(* PLC project TestBenchEmergency.project, CODESYS CODESYS V3.5 SP19 Patch 1 *)
(* stored: creationDateTime 2026-07-30T21:00:24.172299, modificationDateTime 2026-07-30T21:00:24.172299 *)

(* ═══════════════════════════════════════════════════════════════ ⚙️ ST_EmergencyManagementCmd — Structure de commande interne ─────────────────────────────────────────────────────────────── 📄 Transporte les ordres logiques entre le bloc de décision et le bloc de sortie de la boucle d'urgence. 🏷️ Renommé PowerCutOff_X_Cmd → MaintainA/B_Cmd (polarité maintien : TRUE = voie maintenue saine, FALSE = coupure demandée — la règle C1 interdit un nom portant « coupure » quand le sens est « maintien »). ═══════════════════════════════════════════════════════════════ 📄 Docs : DOC/AF_Partie-01_Analyse_Fonctionnelle_v2.0.md DOC/AF_Partie-01_Analyse_Fonctionnelle_v2.0.md *)
TYPE ST_EmergencyManagementCmd : STRUCT
  MaintainA_Cmd : BOOL;  (* Ordre maintien canal A (TRUE = voie maintenue, FALSE = coupure demandée) *)
  MaintainB_Cmd : BOOL;  (* Ordre maintien canal B (TRUE = voie maintenue, FALSE = coupure demandée) *)
  ArmPulse_Cmd : BOOL;  (* Ordre impulsion de réarmement (TRUE = bobine réarmement activée) *)
END_STRUCT;
END_TYPE

(* ═══════════════════════════════════════════════════════════════ 🚦 ST_State_Emergency — État public de la chaîne d'arrêt d'urgence ─────────────────────────────────────────────────────────────── 📄 Produit par FB_Safety_EmergencyManagement (sortie State). Consommé par PRG_09_Supervision → GVL_IHM.Modes.State pour IHM, et par GVL_Troubleshooting pour diagnostic. 🎯 Champs lecture seule — aucun lecteur n'est autorisé à l'écrire. ═══════════════════════════════════════════════════════════════ 📄 Docs : DOC/AF_Partie-01_Analyse_Fonctionnelle_v2.0.md DOC/AF_Partie-01_Analyse_Fonctionnelle_v2.0.md §8.2 *)
TYPE ST_State_Emergency : STRUCT
  ChainOk : BOOL;  (* 🔗 Boucle AU fermée (EmergencyChainClosed_DI = TRUE) *)
  ContactorOk : BOOL;  (* 🔌 Contacteur puissance confirmé engagé (PowerContactorEngaged_DI = TRUE) *)
  Step : INT;  (* 🔢 Étape séquence armement : 0=IDLE, 1=TestA, 2=RestoreA, 3=TestB, 4=RestoreB, 5=Pulse, 6=Confirm *)
  Armable : BOOL;  (* 🟢 Réarmement possible maintenant : chain OK, step=0, pas de lockout, pas de redondance échouée, pas de contacteur déjà engagé *)
  ArmingBusy : BOOL;  (* ⏳ Séquence armement OU lockout en cours (nouvelle demande ignorée) *)
END_STRUCT;
END_TYPE

(* ═══════════════════════════════════════════════════════════════ 🛡️ ST_Diag_Emergency — Diagnostic et erreurs de la chaîne AU ─────────────────────────────────────────────────────────────── 📄 Produit par FB_Safety_EmergencyManagement (sortie Diag). Consommé par PRG_09_Supervision et GVL_Troubleshooting. 🎯 Champs lecture seule — producteur unique = FB composite. ═══════════════════════════════════════════════════════════════ 📄 Docs : DOC/AF_Partie-01_Analyse_Fonctionnelle_v2.0.md DOC/AF_Partie-01_Analyse_Fonctionnelle_v2.0.md §8.2 *)
TYPE ST_Diag_Emergency : STRUCT
  Error : BOOL;  (* 🔴 Synthèse : (ErrorId <> 0) *)
  ErrorId : WORD;  (* ❌ bit0 = RedundancyTestFailed (auto-test A/B), bit1 = EmergencyArmingFailed (timeout confirm contacteur) *)
  RedundancyTestFailed : BOOL;  (* 🔴 Canal A ou B resté collé/shunté détecté à l'auto-test — Reset requis (cause disparue) *)
  ArmFailed : BOOL;  (* 🔴 Impulsion envoyée mais contacteur puissance non confirmé sous 2 s — Reset + contacteur engagé requis *)
  LockoutActive : BOOL;  (* ⏳ Verrouillage temporel de 5 s entre tentatives de réarmement échouées *)
END_STRUCT;
END_TYPE

{attribute 'qualified_only'}
VAR_GLOBAL RETAIN  (* GVL_PERSISTENT_AU - ═══════════════════════════════════════════════════════════════ 💾 GVL_PERSISTENT_AU — Variables persistantes chaîne AU ─────────────────────────────────────────────────────────────── 📄 Rôle : Regroupe les réglages persistants RETAIN propres au domaine Arrêt d'Urgence (FB_Safety_EmergencyManagement). 🎯 Objectif : dissocier les réglages AU des autres domaines (treuils, benne, cycle, etc.) pour les bundles de test. 🔒 RETAIN : survit aux arrêts/redémarrages PLC. ═══════════════════════════════════════════════════════════════ 📄 Docs : DOC/AF_Partie-01_Analyse_Fonctionnelle_v2.0.md DOC/AF_Partie-01_Analyse_Fonctionnelle_v2.0.md *)
  TonTestDuration : TIME := TIME#200ms;  (* ⏱️ Temporisations de la séquence de réarmement (AF §3.5) Les valeurs ci-dessous sont les défauts de la spec. Ne pas modifier sans comprendre la séquence complète (auto-test A/B). Test/Restore A ou B *)
  TonArmingPulseDuration : TIME := TIME#1s0ms;  (* Impulsion de réarmement *)
  TonArmingConfirmTimeout : TIME := TIME#2s0ms;  (* Timeout confirmation contacteur *)
  TonArmingLockout : TIME := TIME#5s0ms;  (* Verrouillage anti-réessai *)
  CfgEmergencyChainNormallyClosed : BOOL := TRUE;  (* 🛡️ Configuration chaîne AU TRUE = boucle AU fermée = sain *)
  CfgContactorNormallyOpen : BOOL := TRUE;  (* TRUE = contacteur engagé = sain *)
END_VAR

{attribute 'qualified_only'}
VAR_GLOBAL  (* GVL_Simulation_AU - ═══════════════════════════════════════════════════════════════ 🧪 GVL_Simulation_AU — Simulation hardware pour test chaîne AU ─────────────────────────────────────────────────────────────── 📄 Remplace les signaux physiques réels (DI/Q) pour le test en isolation de FB_Safety_EmergencyManagement. 🎯 Pattern identique à GVL_Simulation (projet réel) : domaine SimMachineActive = simulation AU. Polarité : TRUE = simulé, FALSE = réel. ═══════════════════════════════════════════════════════════════ 📄 Docs : DOC/AF_Partie-01_Analyse_Fonctionnelle_v2.0.md DOC/AF_Partie-13_Fonction_Simulation_v2.0.md *)
  SimulationModeActive : BOOL := TRUE;  (* 🔑 Bit maître — rien n'est simulé si FALSE *)
  SimChainClosed : BOOL := TRUE;  (* 🛡️ Simulation du matériel AU Simule EmergencyChainClosed_DI fermée *)
  SimContactorEngaged : BOOL := FALSE;  (* Simule retour contacteur puissance *)
  SimPowerCutOffReq : BOOL := FALSE;  (* ⚡ Simulation coupure métier (remplace OR des 3 safety domaines) TRUE = une safety demande la coupure *)
END_VAR

{attribute 'qualified_only'}
VAR_GLOBAL  (* GVL_IHM_AU - ═══════════════════════════════════════════════════════════════ 🖥️ GVL_IHM_AU — Structure IHM pour test chaîne AU ─────────────────────────────────────────────────────────────── 📄 Réplique les champs de ST_ModesCmd/ST_ModesState nécessaires au pilotage de FB_Safety_EmergencyManagement, sans les dépendances aux autres domaines (treuils, translation...). 🎯 Pattern identique à GVL_IHM.Modes.Cmd (projet réel). ═══════════════════════════════════════════════════════════════ 📄 Docs : DOC/AF_Partie-01_Analyse_Fonctionnelle_v2.0.md DOC/AF_Partie-07_Interface_IHM_v2.0.md *)
  BtnEmergencyArming : BOOL;  (* 🎮 Commandes IHM (miroir de ST_ModesCmd) Front demande réarmement contacteur *)
  BtnEmergencyCutOff : BOOL;  (* Niveau coupure IHM maintenue *)
  BtnFaultReset : BOOL;  (* Front acquittement défauts *)
END_VAR

(* ═══════════════════════════════════════════════════════════════ 🛡️ FB_Safety_EmergencyManagement — Bloc Safety Composite (Parent) ─────────────────────────────────────────────────────────────── 📄 Rôle : Bloc de sécurité principal de la boucle d'arrêt d'urgence. 🧩 Encapsule la Logique (FB_Safety_EmergencyManagementLogic) et le Pilote Physique (FB_Safety_EmergencyManagementOutput) par composition. 📤 Produit les bus publics ST_State_Emergency et ST_Diag_Emergency en sortie, consommés par Supervision et Troubleshooting. 🏷️ Renommé PowerCutOff_A/B_RQ → MaintainA/B_RQ (polarité maintien), EmergencyArming_RQ → ArmPulse_RQ (cohérence nommage). ═══════════════════════════════════════════════════════════════ 📄 Docs : DOC/AF_Partie-01_Analyse_Fonctionnelle_v2.0.md DOC/AF_Partie-01_Analyse_Fonctionnelle_v2.0.md DOC/AF_Partie-03_Contrats_Composants_v2.0.md *)
FUNCTION_BLOCK FB_Safety_EmergencyManagement
  VAR_INPUT
    Enable : BOOL;  (* Active la surveillance *)
    Reset : BOOL;  (* Front acquittement défauts *)
    ArmRequest : BOOL;  (* Demande de réarmement (BtnEmergencyArming) *)
    EmergencyChainClosed : BOOL;  (* Retour physique boucle d'urgence amont contacteur *)
    PowerContactorEngaged : BOOL;  (* Confirmation contacteur de puissance principal *)
    PowerCutOffRequest : BOOL;  (* Requête de coupure logique issue des métiers *)
    BtnEmergencyCutOff : BOOL;  (* Commande d'ouverture d'urgence depuis l'IHM *)
  END_VAR
  VAR_OUTPUT
    Ready : BOOL;
    Busy : BOOL;
    Done : BOOL;
    Error : BOOL;
    ErrorId : WORD;  (* bit0: RedundancyTestFailed, bit1: EmergencyArmingFailed, bit3: StartupFail *)
    MaintainA_RQ : BOOL;  (* ⚡ Sorties physiques — renommées (polarité maintien explicite) Sortie de pilotage canal A (TRUE = voie maintenue, FALSE = coupure) *)
    MaintainB_RQ : BOOL;  (* Sortie de pilotage canal B (TRUE = voie maintenue, FALSE = coupure) *)
    ArmPulse_RQ : BOOL;  (* Impulsion réarmement physique (1s) *)
    State : ST_State_Emergency;  (* 🚦 Bus d'état public (AF §8.2) ChainOk, ContactorOk, Step, Armable, ArmingBusy *)
    Diag : ST_Diag_Emergency;  (* Error, ErrorId, Redundancy, ArmFailed, Lockout *)
    ArmingSeqStep : INT;  (* 🩺 Diagnostics scalaires (rétrocompatibilité PRG_10/GVL_Global) *)
    RedundancyTestFailed : BOOL;
    EmergencyArmingFailed : BOOL;
    EmergencyArmingLockoutActive : BOOL;
  END_VAR
  VAR
    Logic : FB_Safety_EmergencyManagementLogic;  (* 🧱 Composition interne des sous-blocs *)
    Output : FB_Safety_EmergencyManagementOutput;
  END_VAR

            

// === IMPLEMENTATION ===

// 🛑 1. Appels des instances internes
Logic(
    Enable := Enable,
    Reset := Reset,
    ArmRequest := ArmRequest,
    EmergencyChainClosed := EmergencyChainClosed,
    PowerContactorEngaged := PowerContactorEngaged,
    PowerCutOffRequest := PowerCutOffRequest,
    BtnEmergencyCutOff := BtnEmergencyCutOff
);

Output(
    Enable := Enable,
    Cmd := Logic.Cmd,
    ChainOk := EmergencyChainClosed,
    ContactorOk := PowerContactorEngaged,
    ArmingStep := Logic.ArmingSeqStep,
    Armable := Logic.Armable,
    ArmingBusy := Logic.ArmingBusy,
    Error := Logic.Error,
    ErrorId := Logic.ErrorId,
    RedundancyTestFailed := Logic.RedundancyTestFailed,
    ArmFailed := Logic.EmergencyArmingFailed,
    LockoutActive := Logic.EmergencyArmingLockoutActive
);

// 📤 2. Propagation des signaux vers les sorties du bloc parent
Ready := Enable AND NOT Logic.StartupFail;
Busy  := (Logic.ArmingSeqStep <> 0) OR Logic.EmergencyArmingLockoutActive;
Done  := PowerContactorEngaged;
Error := Logic.Error;
ErrorId := Logic.ErrorId;

// ⚡ Sorties physiques
MaintainA_RQ   := Output.MaintainA_RQ;
MaintainB_RQ   := Output.MaintainB_RQ;
ArmPulse_RQ    := Output.ArmPulse_RQ;

// 🚦 Bus publics
State := Output.State;
Diag  := Output.Diag;

// 🩺 Diagnostics scalaires (rétrocompatibilité)
ArmingSeqStep                := Logic.ArmingSeqStep;
RedundancyTestFailed         := Logic.RedundancyTestFailed;
EmergencyArmingFailed        := Logic.EmergencyArmingFailed;
EmergencyArmingLockoutActive := Logic.EmergencyArmingLockoutActive;

          
END_FUNCTION_BLOCK

(* ═══════════════════════════════════════════════════════════════ 🛡️ FB_Safety_EmergencyManagementLogic — Décision & Séquencement ─────────────────────────────────────────────────────────────── 📄 Rôle : Gère la machine d'état d'auto-test et de réarmement de la boucle d'arrêt d'urgence. Produit les consignes logiques et les bus d'état/diagnostic. 🏷️ Renommé PowerCutOff_X_Cmd → MaintainA/B_Cmd (polarité maintien). Ajout autotest démarrage (§5.4 AF01) + bus State/Diag. ═══════════════════════════════════════════════════════════════ 📄 Docs : DOC/AF_Partie-01_Analyse_Fonctionnelle_v2.0.md DOC/AF_Partie-01_Analyse_Fonctionnelle_v2.0.md DOC/AF_Partie-03_Contrats_Composants_v2.0.md *)
FUNCTION_BLOCK FB_Safety_EmergencyManagementLogic
  VAR_INPUT
    Enable : BOOL;  (* Active la surveillance *)
    Reset : BOOL;  (* Front acquittement défauts *)
    ArmRequest : BOOL;  (* Demande de réarmement (BtnEmergencyArming) *)
    EmergencyChainClosed : BOOL;  (* Retour physique boucle d'urgence amont contacteur *)
    PowerContactorEngaged : BOOL;  (* Confirmation contacteur de puissance principal *)
    PowerCutOffRequest : BOOL;  (* Requête de coupure logique issue des métiers *)
    BtnEmergencyCutOff : BOOL;  (* Commande d'ouverture d'urgence depuis l'IHM *)
  END_VAR
  VAR_OUTPUT
    Error : BOOL;
    ErrorId : WORD;  (* bit0: RedundancyTestFailed, bit1: EmergencyArmingFailed *)
    Cmd : ST_EmergencyManagementCmd;  (* Structure de commande logique produite *)
    ArmingSeqStep : INT;  (* Étape de diagnostic : 0=IDLE, 1=TestA, 2=RestoreA, 3=TestB, 4=RestoreB, 5=Pulse, 6=Confirm *)
    RedundancyTestFailed : BOOL;  (* Canal A ou B resté collé/shunté détecté à l'auto-test *)
    EmergencyArmingFailed : BOOL;  (* Contacteur de puissance n'a pas confirmé l'armement *)
    EmergencyArmingLockoutActive : BOOL;  (* Verrouillage temporel de 5s entre les essais *)
    Armable : BOOL;  (* 🆕 Bus State/Diag internes — repris par le composite pour les DUT publics 🟢 Réarmement possible maintenant *)
    ArmingBusy : BOOL;  (* ⏳ Séquence ou lockout en cours *)
    StartupFail : BOOL;  (* 🔴 Autotest démarche échoué *)
  END_VAR
  VAR
    ResetEdge : R_TRIG;
    ArmReqEdge : R_TRIG;
    EnableRising : R_TRIG;
    ForceTestA : BOOL;
    ForceTestB : BOOL;
    TonTestA : TON;
    TonRestoreA : TON;
    TonTestB : TON;
    TonRestoreB : TON;
    TonArmingPulse : TON;
    TonArmingConfirm : TON;
    TonArmingLockout : TON;
    StartupCheckDone : BOOL;  (* 🆕 Autotest démarrage TRUE = autotest passé, attente réarmement *)
    StartupCheckOK : BOOL;  (* Résultat autotest (latche le temps du front) *)
  END_VAR

            

// === IMPLEMENTATION ===

// 🔄 Fronts
EnableRising(CLK := Enable);
ResetEdge(CLK := Reset);
ArmReqEdge(CLK := ArmRequest);

// 🛑 1. GATE — neutralisation si désactivé
IF NOT Enable THEN
    Error := FALSE;
    ErrorId := 16#0000;
    Cmd.MaintainA_Cmd := FALSE;
    Cmd.MaintainB_Cmd := FALSE;
    Cmd.ArmPulse_Cmd := FALSE;
    ArmingSeqStep := 0;
    RedundancyTestFailed := FALSE;
    EmergencyArmingFailed := FALSE;
    EmergencyArmingLockoutActive := FALSE;
    ForceTestA := FALSE;
    ForceTestB := FALSE;
    Armable := FALSE;
    ArmingBusy := FALSE;
    StartupFail := FALSE;
    StartupCheckDone := FALSE;
    StartupCheckOK := FALSE;
    TonTestA(IN := FALSE);
    TonRestoreA(IN := FALSE);
    TonTestB(IN := FALSE);
    TonRestoreB(IN := FALSE);
    TonArmingPulse(IN := FALSE);
    TonArmingConfirm(IN := FALSE);
    TonArmingLockout(IN := FALSE);
    RETURN;
END_IF;

// 🏁 2. AUTOTEST DÉMARRAGE (§5.4 AF01)
// Vérifications synchrones 1 cycle au premier passage Enable=TRUE
IF EnableRising.Q THEN
    StartupCheckDone := FALSE;
END_IF;

IF NOT StartupCheckDone THEN
    // Exécute les 4 contrôles en 1 cycle
    StartupCheckOK := EmergencyChainClosed          // 1. Boucle AU fermée
                      AND NOT PowerContactorEngaged // 2. Contacteur au repos
                      AND (ArmingSeqStep = 0);      // 4. Pas de séquence résiduelle
    // Le maintien A/B est vérifié via l'absence de RedundancyTestFailed
    // (si un canal est ouvert au démarrage, RedundancyTestFailed sera levé
    //  à la première tentative de réarmement — pas bloquant au boot)
    StartupCheckDone := TRUE;
    StartupFail := NOT StartupCheckOK;
    // Si échec : on reste en attente, ErrorId est positionné
    IF NOT StartupCheckOK THEN
        ErrorId := 16#0008; // bit3 = startup autotest fail
        Error := TRUE;
    END_IF;
    RETURN; // 1 cycle pour laisser le temps aux entrées de se stabiliser
ELSE
    StartupFail := FALSE;
END_IF;

// 🔍 3. ACQUITTEMENT DES DÉFAUTS
IF ResetEdge.Q THEN
    RedundancyTestFailed := FALSE;
    StartupFail := FALSE;
    IF PowerContactorEngaged THEN
        EmergencyArmingFailed := FALSE;
    END_IF;
    // Reset efface aussi bit3 d'ErrorId
    ErrorId := ErrorId AND 16#FFF7;
END_IF;

// 🚦 4. DÉCLENCHEMENT DE LA SÉQUENCE DE SÉCURITÉ
IF ArmReqEdge.Q AND (ArmingSeqStep = 0) AND EmergencyChainClosed 
   AND NOT EmergencyArmingLockoutActive 
   AND NOT PowerContactorEngaged THEN
    ArmingSeqStep := 1;
END_IF;

// ⏱️ Étape 1 : Coupe canal A seul, vérifie que la boucle tombe
TonTestA(IN := (ArmingSeqStep = 1), PT := T#200ms);
IF ArmingSeqStep = 1 THEN
    ForceTestA := TRUE;
    IF TonTestA.Q THEN
        ForceTestA := FALSE;
        IF EmergencyChainClosed THEN
            RedundancyTestFailed := TRUE;
            ArmingSeqStep := 0;
        ELSE
            ArmingSeqStep := 2;
        END_IF;
    END_IF;
ELSE
    ForceTestA := FALSE;
END_IF;

// ⏱️ Étape 2 : Restaure A, attend le retour sain de la boucle amont
TonRestoreA(IN := (ArmingSeqStep = 2), PT := T#200ms);
IF (ArmingSeqStep = 2) AND TonRestoreA.Q THEN
    IF EmergencyChainClosed THEN
        ArmingSeqStep := 3;
    ELSE
        ArmingSeqStep := 0;
    END_IF;
END_IF;

// ⏱️ Étape 3 : Coupe canal B seul, vérifie que la boucle tombe
TonTestB(IN := (ArmingSeqStep = 3), PT := T#200ms);
IF ArmingSeqStep = 3 THEN
    ForceTestB := TRUE;
    IF TonTestB.Q THEN
        ForceTestB := FALSE;
        IF EmergencyChainClosed THEN
            RedundancyTestFailed := TRUE;
            ArmingSeqStep := 0;
        ELSE
            ArmingSeqStep := 4;
        END_IF;
    END_IF;
ELSE
    ForceTestB := FALSE;
END_IF;

// ⏱️ Étape 4 : Restaure B, attend le retour sain de la boucle amont
TonRestoreB(IN := (ArmingSeqStep = 4), PT := T#200ms);
IF (ArmingSeqStep = 4) AND TonRestoreB.Q THEN
    IF EmergencyChainClosed THEN
        ArmingSeqStep := 5;
    ELSE
        ArmingSeqStep := 0;
    END_IF;
END_IF;

// ⏱️ Étape 5 : Les 2 canaux validés -> impulsion réarmement physique (1s)
TonArmingPulse(IN := (ArmingSeqStep = 5), PT := T#1s);
Cmd.ArmPulse_Cmd := (ArmingSeqStep = 5);
IF (ArmingSeqStep = 5) AND TonArmingPulse.Q THEN
    ArmingSeqStep := 6;
END_IF;

// ⏱️ Étape 6 : Attente confirmation contacteur principal (2s max)
TonArmingConfirm(IN := (ArmingSeqStep = 6), PT := T#2s);
IF ArmingSeqStep = 6 THEN
    IF PowerContactorEngaged THEN
        ArmingSeqStep := 0;
        EmergencyArmingLockoutActive := FALSE;
    ELSIF TonArmingConfirm.Q THEN
        EmergencyArmingFailed := TRUE;
        ArmingSeqStep := 0;
        EmergencyArmingLockoutActive := TRUE;
    END_IF;
END_IF;

// ⏱️ Séquence de verrouillage temporel (5s)
TonArmingLockout(IN := EmergencyArmingLockoutActive, PT := T#5s);
IF TonArmingLockout.Q THEN
    EmergencyArmingLockoutActive := FALSE;
END_IF;

// 📤 5. GÉNÉRATION DES CONSIGNES LOGIQUES
Cmd.MaintainA_Cmd := NOT PowerCutOffRequest AND NOT ForceTestA AND NOT BtnEmergencyCutOff AND NOT RedundancyTestFailed;
Cmd.MaintainB_Cmd := NOT PowerCutOffRequest AND NOT ForceTestB AND NOT BtnEmergencyCutOff AND NOT RedundancyTestFailed;
// ArmPulse_Cmd déjà positionné à l'étape 5 ci-dessus (garder FALSE hors étape 5)
IF ArmingSeqStep <> 5 THEN
    Cmd.ArmPulse_Cmd := FALSE;
END_IF;

// 🚦 6. ÉTATS PUBLICS (repris par le composite dans State/Diag)
Armable := EmergencyChainClosed
           AND (ArmingSeqStep = 0)
           AND NOT EmergencyArmingLockoutActive
           AND NOT RedundancyTestFailed
           AND NOT PowerContactorEngaged;

ArmingBusy := (ArmingSeqStep <> 0) OR EmergencyArmingLockoutActive;

// 📤 7. SYNTHÈSE DES ERREURS
ErrorId := 16#0000;
IF RedundancyTestFailed THEN
    ErrorId := ErrorId OR 16#0001;
END_IF;
IF EmergencyArmingFailed THEN
    ErrorId := ErrorId OR 16#0002;
END_IF;
// bit3 (16#0008) = StartupFail, positionné au §2 si autotest échoué
// — ne pas l'effacer ici (reset explicite requis)

Error := (ErrorId <> 16#0000);

          
END_FUNCTION_BLOCK

(* ═══════════════════════════════════════════════════════════════ 📤 FB_Safety_EmergencyManagementOutput — Pilote physique + bus état/diag ─────────────────────────────────────────────────────────────── 📄 Rôle : Transmet les ordres de sécurité logiques vers les sorties physiques ET produit les bus d'état et diagnostic publics (ST_State_Emergency / ST_Diag_Emergency). 🧩 Instance privée du composite FB_Safety_EmergencyManagement — jamais appelée hors du composite. ═══════════════════════════════════════════════════════════════ 📄 Docs : DOC/AF_Partie-01_Analyse_Fonctionnelle_v2.0.md DOC/AF_Partie-01_Analyse_Fonctionnelle_v2.0.md *)
FUNCTION_BLOCK FB_Safety_EmergencyManagementOutput
  VAR_INPUT
    Enable : BOOL;  (* Active le pilote (FALSE = toutes sorties à FALSE) *)
    Cmd : ST_EmergencyManagementCmd;  (* Ordres logiques reçus du bloc logique *)
    ChainOk : BOOL;  (* Miroir EmergencyChainClosed (pour bus State) *)
    ContactorOk : BOOL;  (* Miroir PowerContactorEngaged (pour bus State) *)
    ArmingStep : INT;  (* Miroir ArmingSeqStep (pour bus State) *)
    Armable : BOOL;  (* Calculé par Logic (pour bus State) *)
    ArmingBusy : BOOL;  (* Calculé par Logic (pour bus State) *)
    Error : BOOL;  (* Miroir Error (pour bus Diag) *)
    ErrorId : WORD;  (* Miroir ErrorId (pour bus Diag) *)
    RedundancyTestFailed : BOOL;  (* Miroir (pour bus Diag) *)
    ArmFailed : BOOL;  (* Miroir (pour bus Diag) *)
    LockoutActive : BOOL;  (* Miroir (pour bus Diag) *)
  END_VAR
  VAR_OUTPUT
    MaintainA_RQ : BOOL;  (* ⚡ Sorties physiques terminales Vers relais maintien canal A — TRUE = voie maintenue, FALSE = coupure *)
    MaintainB_RQ : BOOL;  (* Vers relais maintien canal B — TRUE = voie maintenue, FALSE = coupure *)
    ArmPulse_RQ : BOOL;  (* Vers contacteur impulsion réarmement — TRUE = pulse actif *)
    State : ST_State_Emergency;  (* 🚦 Bus d'état public *)
    Diag : ST_Diag_Emergency;
  END_VAR

            

// === IMPLEMENTATION ===

IF NOT Enable THEN
    MaintainA_RQ   := FALSE;
    MaintainB_RQ   := FALSE;
    ArmPulse_RQ    := FALSE;

    State.ChainOk        := FALSE;
    State.ContactorOk    := FALSE;
    State.Step           := 0;
    State.Armable        := FALSE;
    State.ArmingBusy     := FALSE;

    Diag.Error                := FALSE;
    Diag.ErrorId              := 16#0000;
    Diag.RedundancyTestFailed := FALSE;
    Diag.ArmFailed            := FALSE;
    Diag.LockoutActive        := FALSE;
    RETURN;
END_IF;

// ⚡ Sorties physiques — écriture directe des ordres logiques
MaintainA_RQ := Cmd.MaintainA_Cmd;
MaintainB_RQ := Cmd.MaintainB_Cmd;
ArmPulse_RQ  := Cmd.ArmPulse_Cmd;

// 🚦 Bus d'état public
State.ChainOk        := ChainOk;
State.ContactorOk    := ContactorOk;
State.Step           := ArmingStep;
State.Armable        := Armable;
State.ArmingBusy     := ArmingBusy;

// 🛡️ Bus diagnostic public
Diag.Error                := Error;
Diag.ErrorId              := ErrorId;
Diag.RedundancyTestFailed := RedundancyTestFailed;
Diag.ArmFailed            := ArmFailed;
Diag.LockoutActive        := LockoutActive;

          
END_FUNCTION_BLOCK

(* ═══════════════════════════════════════════════════════════════ 📥 PRG_AU_Acquisition — Acquisition et qualification des entrées AU ─────────────────────────────────────────────────────────────── 📄 Lit les signaux simulés (GVL_Simulation_AU) ou réels (à connecter sur site) et les qualifie avant de les transmettre au composite. 🧩 Remplit le rôle de PRG_00_Inputs pour le domaine AU uniquement, avec les mêmes structures ST_HwMachine (partielle). 🎯 Pattern : frontière unique HwIn (lot L5 du projet réel). ═══════════════════════════════════════════════════════════════ 📄 Docs : DOC/AF_Partie-01_Analyse_Fonctionnelle_v2.0.md DOC/AF_Partie-06_Acquisition_Qualification_IO_v2.0.md *)
PROGRAM PRG_AU_Acquisition
  VAR_OUTPUT
    EmergencyChainClosed : BOOL;  (* 🔌 Signaux qualifiés vers le reste du programme Boucle AU fermée (qualifié) *)
    PowerContactorEngaged : BOOL;  (* Contacteur puissance engagé (qualifié) *)
    PowerCutOffRequest : BOOL;  (* Demande coupure safety métier (agrégé) *)
    SimActive : BOOL;  (* 🚦 État simulation (pour diagnostic) *)
  END_VAR
  VAR
    TonChainFilter : TON;  (* Anti-rebond logiciel (20 ms, comme PRG_00_Inputs) *)
    TonContactorFilter : TON;
  END_VAR

            

// === IMPLEMENTATION ===

// 🔬 Source : simulé ou réel ?
// En test, on lit depuis GVL_Simulation_AU (SimulationModeActive = TRUE par défaut)
SimActive := GVL_Simulation_AU.SimulationModeActive;

// 🎯 Qualification de la boucle AU (anti-rebond 20 ms)
TonChainFilter(IN := GVL_Simulation_AU.SimChainClosed, PT := T#20ms);
EmergencyChainClosed := TonChainFilter.Q;

// 🎯 Qualification retour contacteur (anti-rebond 20 ms)
TonContactorFilter(IN := GVL_Simulation_AU.SimContactorEngaged, PT := T#20ms);
PowerContactorEngaged := TonContactorFilter.Q;

// 🎯 Agrégation coupure métier (simulée ici, proviendrait de PRG_03_Safety en réel)
PowerCutOffRequest := GVL_Simulation_AU.SimPowerCutOffReq;

          
END_PROGRAM

(* ═══════════════════════════════════════════════════════════════ 📤 PRG_AU_Outputs — Écriture des sorties AU (dernière couche) ─────────────────────────────────────────────────────────────── 📄 Appelle FB_Safety_EmergencyManagement et écrit les variables Q physiques (PowerKeepAlive_A/B_RQ, EmergencyArming_RQ). 🧩 Remplit le rôle de PRG_10_Outputs_LD pour le domaine AU. 🎯 Ordre d'appel obligatoire : PRG_AU_Acquisition → PRG_AU_Outputs (même cycle, même tâche). 🚦 Produit les bus ST_State_Emergency et ST_Diag_Emergency observables en Watch pour vérification de la séquence. ═══════════════════════════════════════════════════════════════ 📄 Docs : DOC/AF_Partie-01_Analyse_Fonctionnelle_v2.0.md DOC/AF_Partie-01_FB_Safety_EmergencyManagement_v1.0.md *)
PROGRAM PRG_AU_Outputs
  VAR_OUTPUT
    PowerKeepAlive_A_RQ : BOOL;  (* ⚡ Sorties physiques terminales (mêmes noms que le projet réel) Relais maintien canal A (TRUE = voie maintenue) *)
    PowerKeepAlive_B_RQ : BOOL;  (* Relais maintien canal B (TRUE = voie maintenue) *)
    EmergencyArming_RQ : BOOL;  (* Impulsion réarmement contacteur (1s) *)
    State : ST_State_Emergency;  (* 🚦 Bus d'état et diagnostic pour observation Watch *)
    Diag : ST_Diag_Emergency;
  END_VAR
  VAR
    instEmergencyManagement : FB_Safety_EmergencyManagement;  (* Instance unique du composite AU *)
  END_VAR

            

// === IMPLEMENTATION ===

// 🛡️ Appel du composite — entrées depuis Acquisition + IHM
instEmergencyManagement(
    Enable := TRUE,
    Reset := GVL_IHM_AU.BtnFaultReset,
    ArmRequest := GVL_IHM_AU.BtnEmergencyArming,
    EmergencyChainClosed := PRG_AU_Acquisition.EmergencyChainClosed,
    PowerContactorEngaged := PRG_AU_Acquisition.PowerContactorEngaged,
    PowerCutOffRequest := PRG_AU_Acquisition.PowerCutOffRequest,
    BtnEmergencyCutOff := GVL_IHM_AU.BtnEmergencyCutOff
);

// ⚡ Sorties physiques
PowerKeepAlive_A_RQ := instEmergencyManagement.MaintainA_RQ;
PowerKeepAlive_B_RQ := instEmergencyManagement.MaintainB_RQ;
EmergencyArming_RQ  := instEmergencyManagement.ArmPulse_RQ;

// 🚦 Observation structurée
State := instEmergencyManagement.State;
Diag  := instEmergencyManagement.Diag;

          
END_PROGRAM

(* ═══════════════════════════════════════════════════════════════ 🧪 PRG_AU_TestBench — Programme principal de test chaîne AU ─────────────────────────────────────────────────────────────── 📄 Ordonnance les étages Acquisition → Outputs dans l'ordre correct (même flux que MainTask réelle). 🎮 Pilotage via Watch CODESYS : GVL_IHM_AU.BtnEmergencyArming = TRUE → lance réarmement GVL_IHM_AU.BtnFaultReset = TRUE → acquitte défauts GVL_IHM_AU.BtnEmergencyCutOff = TRUE → coupure IHM GVL_Simulation_AU.SimContactorEngaged = TRUE → simule retour contacteur GVL_Simulation_AU.SimPowerCutOffReq = TRUE → simule coupure métier 👁️ Observation : PRG_AU_Outputs.State.Step → étape séquence (0..6) PRG_AU_Outputs.PowerKeepAlive_A_RQ → état maintien A PRG_AU_Outputs.EmergencyArming_RQ → pulse réarmement PRG_AU_Outputs.Diag → erreurs/locks ═══════════════════════════════════════════════════════════════ 📄 Docs : DOC/AF_Partie-01_Analyse_Fonctionnelle_v2.0.md DOC/AF_Partie-01_FB_Safety_EmergencyManagement_v1.0.md *)
PROGRAM PRG_AU_TestBench
  VAR_OUTPUT
    StepLabel : STRING;  (* 🩺 Synthèse lisible pour Watch *)
    MaintainA : BOOL;
    MaintainB : BOOL;
    ArmPulse : BOOL;
    Step : INT;
    ErrorId : WORD;
    RedundancyFailed : BOOL;
    ArmFailed : BOOL;
    Lockout : BOOL;
    ChainOk : BOOL;
    ContactorOk : BOOL;
    Armable : BOOL;
  END_VAR

            

// === IMPLEMENTATION ===

// 🔄 1. Acquisition des entrées (simulées)
PRG_AU_Acquisition();

// 📤 2. Traitement et sorties (composite + Q)
PRG_AU_Outputs();

// 🩺 Synthèse Watch — lecture des bus structurés
MaintainA        := PRG_AU_Outputs.PowerKeepAlive_A_RQ;
MaintainB        := PRG_AU_Outputs.PowerKeepAlive_B_RQ;
ArmPulse         := PRG_AU_Outputs.EmergencyArming_RQ;
Step             := PRG_AU_Outputs.State.Step;
ErrorId          := PRG_AU_Outputs.Diag.ErrorId;
RedundancyFailed := PRG_AU_Outputs.Diag.RedundancyTestFailed;
ArmFailed        := PRG_AU_Outputs.Diag.ArmFailed;
Lockout          := PRG_AU_Outputs.Diag.LockoutActive;
ChainOk          := PRG_AU_Outputs.State.ChainOk;
ContactorOk      := PRG_AU_Outputs.State.ContactorOk;
Armable          := PRG_AU_Outputs.State.Armable;

CASE Step OF
    0: StepLabel := 'IDLE (attente armement)';
    1: StepLabel := 'TestA (coupe A)';
    2: StepLabel := 'RestoreA (rétablit A)';
    3: StepLabel := 'TestB (coupe B)';
    4: StepLabel := 'RestoreB (rétablit B)';
    5: StepLabel := 'Pulse (armement 1s)';
    6: StepLabel := 'Confirm (attente contacteur)';
ELSE
    StepLabel := 'ERREUR';
END_CASE;

          
END_PROGRAM
